// TIA Portal project "encoder 5" (V16)

(* hardware
DEVICE "S7-1200 station_1"  S7-1200 Station
   slot 0: "Rack_0"  S7-1200 Rack  Rack  V1.0
   slot 1: "PLC_1"  CPU 1212C DC/DC/DC  6ES7 212-1AE40-0XB0  V4.1
*)

// ===== PLC "PLC_1"  CPU 1212C DC/DC/DC =====

VAR_GLOBAL   // PLC tag table "Default tag table"
   "ATIVA MOTOR_BK10_2201" AT %M0.0 : Bool;
   "ATIVA_MOTOR_BK10_2201" AT %Q0.0 : Bool;
   "AUT/MAN_BK10_2201" AT %I0.2 : Bool;
   "ENCODER VERDE A_BK10_2201" AT %I0.0 : Bool;
   "ENCODER_BK10_2201" AT %ID1000 : DInt;
   "SINALEIRO_BK10_2201" AT %Q0.1 : Bool;
   "ATIVA MOTOR_BK10_2301" AT %M0.1 : Bool;
   "ATIVA_MOTOR_BK10_2301" AT %Q0.2 : Bool;
   "AUT/MAN_BK10_2301" AT %I0.3 : Bool;
   "ENCODER2 VERDE A_BK10_2301" AT %I0.1 : Bool;
   "ENCODER_BK10_2301" AT %ID1004 : DInt;
   "SINALEIRO_BK10_2301" AT %Q0.3 : Bool;
   "liga_motor_manual_BK10_2201" AT %I0.4 : Bool;
   "liga_motor_manual_BK10_2301" AT %I0.5 : Bool;
END_VAR

// folder: System blocks/Program resources

DATA_BLOCK "IEC_Timer_0_DB"   // DB2
{ S7_Optimized_Access := 'TRUE' }
AUTHOR : Simatic
FAMILY : IEC
NAME : IEC_TMR
VERSION : 1.0
// stored: InstanceOfName IEC_TIMER
"IEC_TIMER"
BEGIN
END_DATA_BLOCK

DATA_BLOCK "DB_ENCODER_2301"   // DB5
{ S7_Optimized_Access := 'TRUE' }
AUTHOR : Simatic
FAMILY : IEC
NAME : IEC_TMR
VERSION : 1.0
// stored: InstanceOfName IEC_TIMER
"IEC_TIMER"
BEGIN
END_DATA_BLOCK

// folder: (top level)

ORGANIZATION_BLOCK "OB_BK10_2201"   // OB1, LAD, ProgramCycle
TITLE = "Main Program Sweep (Cycle)"
{ S7_Optimized_Access := 'TRUE' }
VERSION : 0.1
   VAR_INPUT
      Initial_Call : Bool;   // Initial call of this OB
      Remanence : Bool;   // =True, if remanent data are available
   END_VAR
   VAR_TEMP
      Temp_1 : Bool;
   END_VAR
BEGIN

REGION Network 1
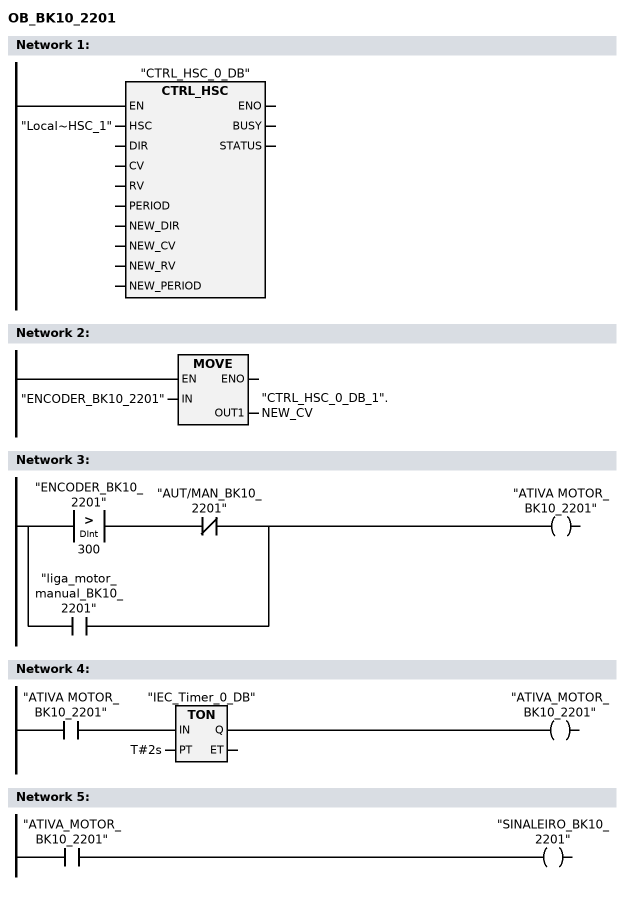
   "CTRL_HSC_0_DB"(HSC := "Local~HSC_1");   // CTRL_HSC
END_REGION

REGION Network 2
   RUNG wire#powerrail
      Move(in := "ENCODER_BK10_2201", out1 => "CTRL_HSC_0_DB_1".NEW_CV)
   END_RUNG
   // the same network as SCL:
   "CTRL_HSC_0_DB_1".NEW_CV := "ENCODER_BK10_2201";
END_REGION

REGION Network 3
   RUNG wire#powerrail
      { S7_Templates := "SrcType := DInt" } GT_Contact(in1 := "ENCODER_BK10_2201", in2 := 300)
      I_Contact( "AUT/MAN_BK10_2201" )
      wire#w1
      Coil( "ATIVA MOTOR_BK10_2201" )
   END_RUNG
   RUNG wire#powerrail
      Contact( "liga_motor_manual_BK10_2201" )
   END_RUNG wire#w1
   // the same network as SCL:
   "ATIVA MOTOR_BK10_2201" := (("ENCODER_BK10_2201" > 300) AND NOT "AUT/MAN_BK10_2201") OR "liga_motor_manual_BK10_2201";
END_REGION

REGION Network 4
   "IEC_Timer_0_DB".TON(IN := "ATIVA MOTOR_BK10_2201", PT := T#2s);
   "ATIVA_MOTOR_BK10_2201" := "IEC_Timer_0_DB".Q;
END_REGION

REGION Network 5
   RUNG wire#powerrail
      Contact( "ATIVA_MOTOR_BK10_2201" )
      Coil( "SINALEIRO_BK10_2201" )
   END_RUNG
   // the same network as SCL:
   "SINALEIRO_BK10_2201" := "ATIVA_MOTOR_BK10_2201";
END_REGION
END_ORGANIZATION_BLOCK

ORGANIZATION_BLOCK "OB_BK10_2301"   // OB123, LAD, ProgramCycle
TITLE = "Main Program Sweep (Cycle)"
{ S7_Optimized_Access := 'TRUE' }
VERSION : 0.1
   VAR_INPUT
      Initial_Call : Bool;   // Initial call of this OB
      Remanence : Bool;   // =True, if remanent data are available
   END_VAR
BEGIN

REGION Network 1
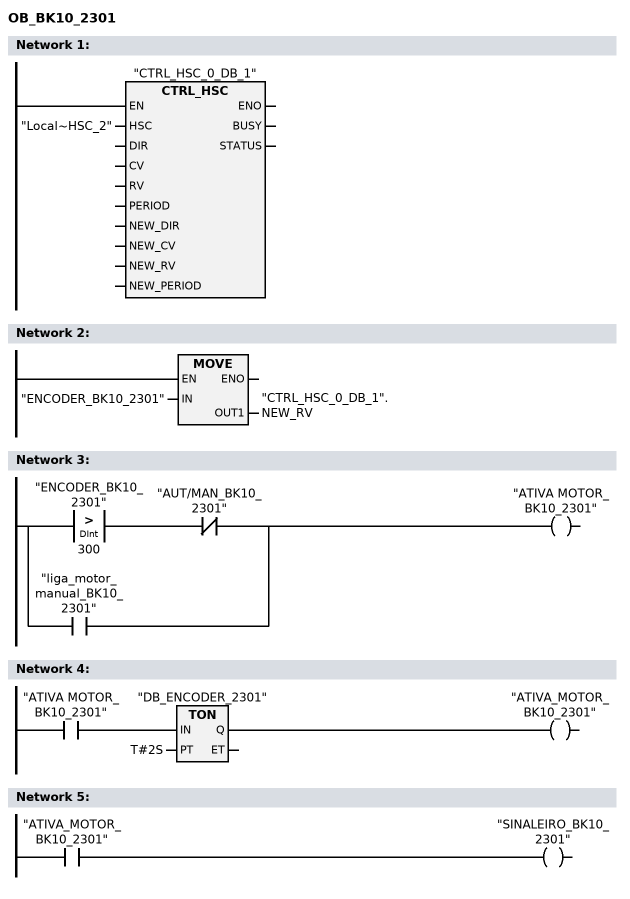
   "CTRL_HSC_0_DB_1"(HSC := "Local~HSC_2");   // CTRL_HSC
END_REGION

REGION Network 2
   RUNG wire#powerrail
      Move(in := "ENCODER_BK10_2301", out1 => "CTRL_HSC_0_DB_1".NEW_RV)
   END_RUNG
   // the same network as SCL:
   "CTRL_HSC_0_DB_1".NEW_RV := "ENCODER_BK10_2301";
END_REGION

REGION Network 3
   RUNG wire#powerrail
      { S7_Templates := "SrcType := DInt" } GT_Contact(in1 := "ENCODER_BK10_2301", in2 := 300)
      I_Contact( "AUT/MAN_BK10_2301" )
      wire#w1
      Coil( "ATIVA MOTOR_BK10_2301" )
   END_RUNG
   RUNG wire#powerrail
      Contact( "liga_motor_manual_BK10_2301" )
   END_RUNG wire#w1
   // the same network as SCL:
   "ATIVA MOTOR_BK10_2301" := (("ENCODER_BK10_2301" > 300) AND NOT "AUT/MAN_BK10_2301") OR "liga_motor_manual_BK10_2301";
END_REGION

REGION Network 4
   "DB_ENCODER_2301".TON(IN := "ATIVA MOTOR_BK10_2301", PT := T#2S);
   "ATIVA_MOTOR_BK10_2301" := "DB_ENCODER_2301".Q;
END_REGION

REGION Network 5
   RUNG wire#powerrail
      Contact( "ATIVA_MOTOR_BK10_2301" )
      Coil( "SINALEIRO_BK10_2301" )
   END_RUNG
   // the same network as SCL:
   "SINALEIRO_BK10_2301" := "ATIVA_MOTOR_BK10_2301";
END_REGION
END_ORGANIZATION_BLOCK